(* PLC project capteur_tor, TNI-Software ControlBuild 4.00 *)
(* stored: creationDateTime 2018-09-17T15:33:38-01:00 *)

CONFIGURATION capteur_tor
  VAR_GLOBAL
    simuperiod : REAL := 50000.0;
    taskname : STRING(50) := 'capteur_tor.exe';
    allowpreconditions : BOOL := true;
    allowpostconditions : BOOL := true;
  END_VAR
END_CONFIGURATION
